Fanuc KAREL source: kt00160.KL

-- PROVISIONAL review KL for V940-1; original PC SHA256 065bb1ba2d85d19b49831e01ffc818962ef154916a949e562bc78d1074f0cc67
-- Incomplete behavior may be omitted. Consult companion uncertainty JSON. Do not deploy.
PROGRAM KT00160
%NOLOCKGROUP
VAR
  OUT : REAL
-- UNRESOLVED_DECL H1 type=002017
-- UNRESOLVED_DECL H2 type=002017
BEGIN
  -- V9_ZERO_TABLE_METADATA_HINT layout=0001; no indexed target words; source/name/runtime held
  -- UNRESOLVED_PC offsets 5-19; opcodes 2E,22,9D,33,B4
  -- UNRESOLVED_PC offsets 24-38; opcodes 2E,22,9D,33,B4
  -- UNRESOLVED_PC offsets 43-57; opcodes 2E,22,9D,33,B4
  -- UNRESOLVED_PC offsets 62-76; opcodes 2E,22,9D,33,B4
  -- UNRESOLVED_PC offsets 81-107; opcodes 22,9D,33,B3,22,9D,33,B3,55,64,23
  -- UNRESOLVED_PC offsets 112-116; opcodes 7F
END KT00160
